INTERFACE I_Base EXTENDS I_Object, I_FastCall, I_MainCall

END_INTERFACE

(* stored: Version 1.1.0.1
   Itf I_Base: Id {70e0496d-fdea-401d-8bb5-41f0b622480f} *)
